(* IEC 61131-3 sources: CodesysTest/alpha/export/Device.dev/Plc Logic/Application/FBs/DataHandlers/ModbusLongHandlerFB.pou, 2 files *)

(* ---- ModbusLongHandlerFB.pou.st ---- *)
(*#-#-#-#-#-#-#-#-#-#---Declaration---#-#-#-#-#-#-#-#-#-#-#-#-#*)

FUNCTION_BLOCK ModbusLongHandlerFB
VAR_INPUT
    modbusLong : ModbusLongType;
END_VAR
VAR_OUTPUT
END_VAR
VAR
END_VAR(*#-#-#-#-#-#-#-#-#-#---Implementation---#-#-#-#-#-#-#-#-#-#-#-#-#*)

(* ---- Pack.m.st ---- *)
(*#-#-#-#-#-#-#-#-#-#---Declaration---#-#-#-#-#-#-#-#-#-#-#-#-#*)

METHOD Pack
VAR_IN_OUT
    modbusLong : ModbusLongType;
END_VAR
(*#-#-#-#-#-#-#-#-#-#---Implementation---#-#-#-#-#-#-#-#-#-#-#-#-#*)

modbusLong.rawValue := DWORD_TO_DINT(OSCAT_BASIC.DWORD_OF_WORD(modbusLong.highWord,modbusLong.lowWord));
